KUKA KRL program: UP1.src, UP1.dat

--- UP1.src ---
&ACCESS RVP
&REL 1
&COMMENT Auto-loop PTP Move to P1 with external trigger
DEF SIMPLE_MOVE ( )
    ; Initialize the program
    BAS (#INITMOV, 0)

    ; Set motion parameters
    $VEL.CP = 0.25      ; Set velocity to 25% of maximum
    $ACC.CP = 50        ; Set acceleration to 50%
    $APO.CPTP = 100     ; Set approximation distance for PTP motion

    ; Main loop: wait for trigger and move to P1
    LOOP
        ; Wait for external trigger (e.g., $IN[1] set by KUKAVARPROXY)
        WAIT FOR TRIG_USER

        ; Move to position P1
        PTP P1

        ; Optional: Wait for trigger to be reset before next cycle
        WAIT FOR NOT TRIG_USER
    ENDLOOP

    ; End of program
END

--- UP1.dat ---
&ACCESS RVP
&REL 1
&COMMENT Auto-loop PTP Move to P1 with external trigger
DEFDAT SIMPLE_MOVE

; Define position P1
DECL E6POS P1={x 309.227112,y -149.653107,z 1745.69702,a -77.6270523,b -57.8837891,c -160.023407,s 2,t 34,e1 0.0,e2 0.0,e3 0.0,e4 0.0,e5 0.0,e6 0.0}

ENDDAT
